// TIA Portal V20 export
FUNCTION_BLOCK "CallGeneral"   // FB48, LAD
TITLE = CallGeneral
{ S7_Optimized_Access := 'TRUE' }
// General functionality is called in this block. That includes blocks to generate system data as well as blocks that connect handle multiple HMIs.
// stored: IsIECCheckEnabled true, MemoryReserve 100, SetENOAutomatically true
   VAR
      statClockByteOld { ExternalWritable := 'False'} : Byte;   // Stored clock byte from last cycle for rising edge detection
      instLAF_PowerOnOff { ExternalWritable := 'False'} : "LAF_PowerOnOff";
      instLAF_ClockGen { ExternalWritable := 'False'} : "LAF_ClockGenerator";
      instLSNTP_Server { ExternalWritable := 'False'} : "LSNTP_Server";
      instHmiManager { ExternalWritable := 'False'} : "LAF_HmiHeaderSingleUnitManager";
   END_VAR
   VAR_TEMP
      tempIndex : DInt;   // Temp variable for for-loop
      tempHeaderConfig : "LUC_typeHeaderConfig";
      tempAcknowledgeFromHmi : Bool;   // Summarized acknowledge command
      tempPowerOffFromHmi : Bool;   // Summarized power off command
      tempPowerOnFromHmi : Bool;   // Summarized power on command
      tempPowerStatus : Int;   // 0 - Off, 1 - Paused, 2 - On
      tempResultXor : Byte;   // Interim result of XOR operation
      tempPosPulse : Byte;   // Interim result puls calculation
      tempRetValLocT : Int;   // Return value of RD_LOC_T
      tempUpperBoundUnits : DInt;   // Upper bound of unitInterface array for loop execution
   END_VAR
   VAR CONSTANT
      RESET_BUTTON__COULD_BE_ADDED_HERE : Bool := false;   // Placeholder for a potential global reset button
      DAYLIGHT_SAVING_TIME : Int := 1;   // Local time is output as daylight saving time
   END_VAR
   VAR_TEMP   // added for the SCL form of the ladder/FBD networks
      _w1 : Bool;
   END_VAR
BEGIN

REGION Network 1 (SCL): Set visibility of buttons in header popups
   // This code is executed just in the first cycle after all units have published their state machine config in the unit interface during their own Startup OBs.
   //Execute the code just in the first cycle
   IF "Data".general.firstCycle THEN

       //Initialize temp variables
       #tempHeaderConfig.modeButtonsVisibility :=
       #tempHeaderConfig.stateButtonsVisibility :=
       #tempHeaderConfig.specialFunctionButtonsVisibility := 16#0;

       //Loop through the units and summarize enabled modes, states and special functions
       FOR #tempIndex := 0 TO "NO_OF_UNITS" DO
           #tempHeaderConfig.modeButtonsVisibility := #tempHeaderConfig.modeButtonsVisibility OR "Units".unit[#tempIndex].stateMachine.enabledModes;
           #tempHeaderConfig.stateButtonsVisibility := #tempHeaderConfig.stateButtonsVisibility OR "Units".unit[#tempIndex].stateMachine.enabledStates;
           #tempHeaderConfig.specialFunctionButtonsVisibility := #tempHeaderConfig.specialFunctionButtonsVisibility OR "Units".unit[#tempIndex].stateMachine.enabledSpecialFunctions;
       END_FOR;

       //Write summary to config of HMI header
       "Hmi".headerConfig := #tempHeaderConfig;
   END_IF;
END_REGION

REGION Network 2 (SCL): Summarize HMI commands from different panels
   // Read commands for acknowledge, powerOn and powerOff from the different HMI panels and summarize them in temp variables for further logic in this block.
   // Initialize temp variables
   #tempAcknowledgeFromHmi :=
   #tempPowerOffFromHmi :=
   #tempPowerOnFromHmi := FALSE;

   // Loop through the HMI panels and summarize the commands
   FOR #tempIndex := 0 TO "NO_OF_HMI_PANELS" DO
       #tempAcknowledgeFromHmi := #tempAcknowledgeFromHmi OR "Hmi".mainHeader[#tempIndex].hmiToPlc.acknowledge;
       #tempPowerOffFromHmi := #tempPowerOffFromHmi OR "Hmi".mainHeader[#tempIndex].hmiToPlc.powerCommands.%X0;
       #tempPowerOnFromHmi := #tempPowerOnFromHmi OR "Hmi".mainHeader[#tempIndex].hmiToPlc.powerCommands.%X1;
   END_FOR;
END_REGION

REGION Network 3: Global Acknowledge
   // The global acknowledge command from the hmi button is assigned to Global.Data.general.acknowledge: This bit it forwarded to all underlaying modules
   // If a hard-wired global reset button exists, it can
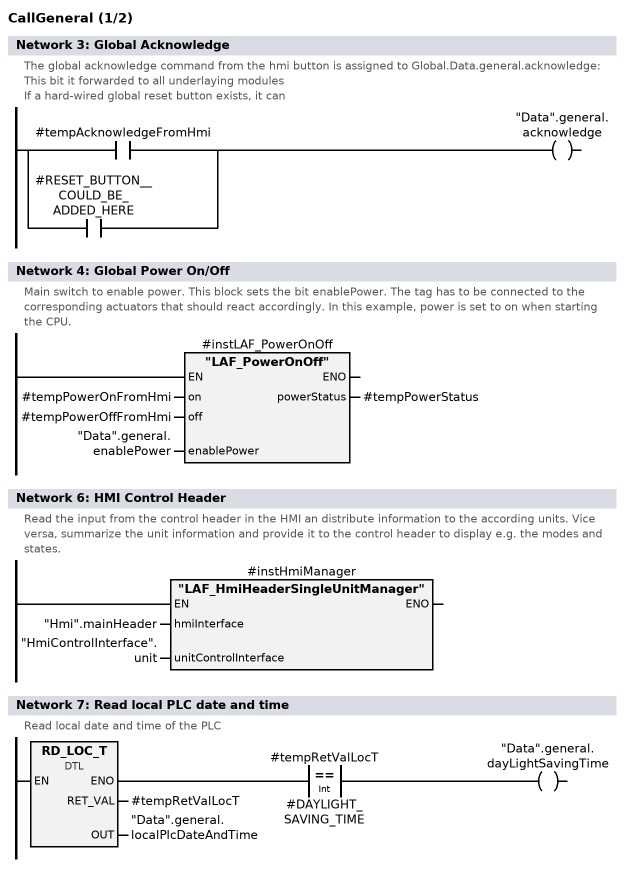
   RUNG wire#powerrail
      Contact( #tempAcknowledgeFromHmi )
      wire#w1
      Coil( "Data".general.acknowledge )
   END_RUNG
   RUNG wire#powerrail
      Contact( #RESET_BUTTON__COULD_BE_ADDED_HERE )
   END_RUNG wire#w1
   // the same network as SCL:
   "Data".general.acknowledge := #tempAcknowledgeFromHmi OR #RESET_BUTTON__COULD_BE_ADDED_HERE;
END_REGION

REGION Network 4: Global Power On/Off
   // Main switch to enable power. This block sets the bit enablePower. The tag has to be connected to the corresponding actuators that should react accordingly. In this example, power is set to on when starting the CPU.
   RUNG wire#powerrail
      #instLAF_PowerOnOff(on := #tempPowerOnFromHmi, off := #tempPowerOffFromHmi, enablePower := "Data".general.enablePower, powerStatus => #tempPowerStatus)
   END_RUNG
   // the same network as SCL:
   #instLAF_PowerOnOff(on := #tempPowerOnFromHmi,   // "LAF_PowerOnOff"
                       off := #tempPowerOffFromHmi,
                       enablePower := "Data".general.enablePower,
                       powerStatus => #tempPowerStatus);
END_REGION

REGION Network 5 (SCL): Write power status to HMI panels
   // Write power status back to all connected HMI panels
   // Loop through the panels and set the power status
   FOR #tempIndex := 0 TO "NO_OF_HMI_PANELS" DO
       "Hmi".mainHeader[#tempIndex].plcToHmi.powerStatus := #tempPowerStatus;
   END_FOR;
END_REGION

REGION Network 6: HMI Control Header
   // Read the input from the control header in the HMI an distribute information to the according units. Vice versa, summarize the unit information and provide it to the control header to display e.g. the modes and states.
   RUNG wire#powerrail
      #instHmiManager(hmiInterface := "Hmi".mainHeader, unitControlInterface := "HmiControlInterface".unit)
   END_RUNG
   // the same network as SCL:
   #instHmiManager(hmiInterface := "Hmi".mainHeader, unitControlInterface := "HmiControlInterface".unit);   // "LAF_HmiHeaderSingleUnitManager"
END_REGION

REGION Network 7: Read local PLC date and time
   // Read local date and time of the PLC
   RUNG wire#powerrail
      { S7_Templates := "date_type := DTL" } RD_LOC_T(RET_VAL => #tempRetValLocT, OUT => "Data".general.localPlcDateAndTime)
      { S7_Templates := "SrcType := Int" } EQ_Contact(in1 := #tempRetValLocT, in2 := #DAYLIGHT_SAVING_TIME)
      Coil( "Data".general.dayLightSavingTime )
   END_RUNG
   // the same network as SCL:
   #tempRetValLocT := RD_LOC_T(OUT => "Data".general.localPlcDateAndTime, ENO => #_w1);
   "Data".general.dayLightSavingTime := #_w1 AND (#tempRetValLocT = #DAYLIGHT_SAVING_TIME);
END_REGION

REGION Network 8: Create clock bits
   // The clock bits are generated instead of the HW clock memory byte of the PLC. Due to the use of software units, the ussage of system and clock memory bytes isn't possible.
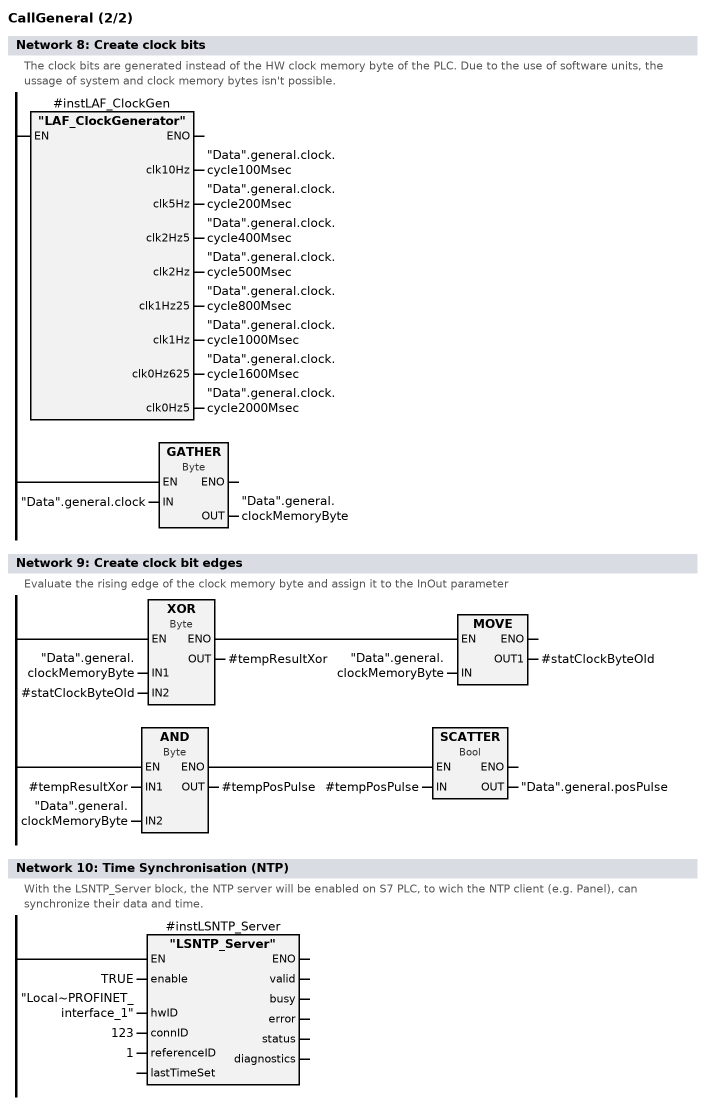
   RUNG wire#powerrail
      #instLAF_ClockGen(clk10Hz => "Data".general.clock.cycle100Msec, clk5Hz => "Data".general.clock.cycle200Msec, clk2Hz5 => "Data".general.clock.cycle400Msec, clk2Hz => "Data".general.clock.cycle500Msec, clk1Hz25 => "Data".general.clock.cycle800Msec, clk1Hz => "Data".general.clock.cycle1000Msec, clk0Hz625 => "Data".general.clock.cycle1600Msec, clk0Hz5 => "Data".general.clock.cycle2000Msec)
   END_RUNG
   RUNG wire#powerrail
      { S7_Templates := "[dest_type := Byte, src_type := Bool]" } GATHER(IN := "Data".general.clock, OUT => "Data".general.clockMemoryByte)
   END_RUNG
   // the same network as SCL:
   #instLAF_ClockGen(clk10Hz => "Data".general.clock.cycle100Msec,   // "LAF_ClockGenerator"
                     clk5Hz => "Data".general.clock.cycle200Msec,
                     clk2Hz5 => "Data".general.clock.cycle400Msec,
                     clk2Hz => "Data".general.clock.cycle500Msec,
                     clk1Hz25 => "Data".general.clock.cycle800Msec,
                     clk1Hz => "Data".general.clock.cycle1000Msec,
                     clk0Hz625 => "Data".general.clock.cycle1600Msec,
                     clk0Hz5 => "Data".general.clock.cycle2000Msec);
   GATHER(IN := "Data".general.clock, OUT => "Data".general.clockMemoryByte);
END_REGION

REGION Network 9: Create clock bit edges
   // Evaluate the rising edge of the clock memory byte and assign it to the InOut parameter
   #tempResultXor := "Data".general.clockMemoryByte XOR #statClockByteOld;
   #statClockByteOld := "Data".general.clockMemoryByte;
   #tempPosPulse := #tempResultXor AND "Data".general.clockMemoryByte;
   SCATTER(IN := #tempPosPulse, OUT => "Data".general.posPulse);
END_REGION

REGION Network 10: Time Synchronisation (NTP)
   // With the LSNTP_Server block, the NTP server will be enabled on S7 PLC, to wich the NTP client (e.g. Panel), can synchronize their data and time.
   RUNG wire#powerrail
      #instLSNTP_Server(enable := TRUE, hwID := "Local~PROFINET_interface_1", connID := 123, referenceID := 1, lastTimeSet :=, valid =>, busy =>, error =>, status =>, diagnostics =>)
   END_RUNG
   // the same network as SCL:
   #instLSNTP_Server(enable := TRUE, hwID := "Local~PROFINET_interface_1", connID := 123, referenceID := 1);   // "LSNTP_Server"
END_REGION
END_FUNCTION_BLOCK
